PROGRAM main
  VAR
    objectDetected AT %IX0.0 : BOOL;
    heightReading AT %IW0 : INT;
    conveyorRun AT %QX0.0 : BOOL;
    diverterGate AT %QX0.1 : BOOL;
    alarmActive AT %QX0.2 : BOOL;
    startCmd AT %QX0.3 : BOOL;
    stopCmd AT %QX0.4 : BOOL;
    resetCmd AT %QX0.5 : BOOL;
    systemRunning AT %QX0.6 : BOOL;
    isTallObject : BOOL;
    TON0 : TON;
    TON1 : TON;
    h : REAL;
  END_VAR

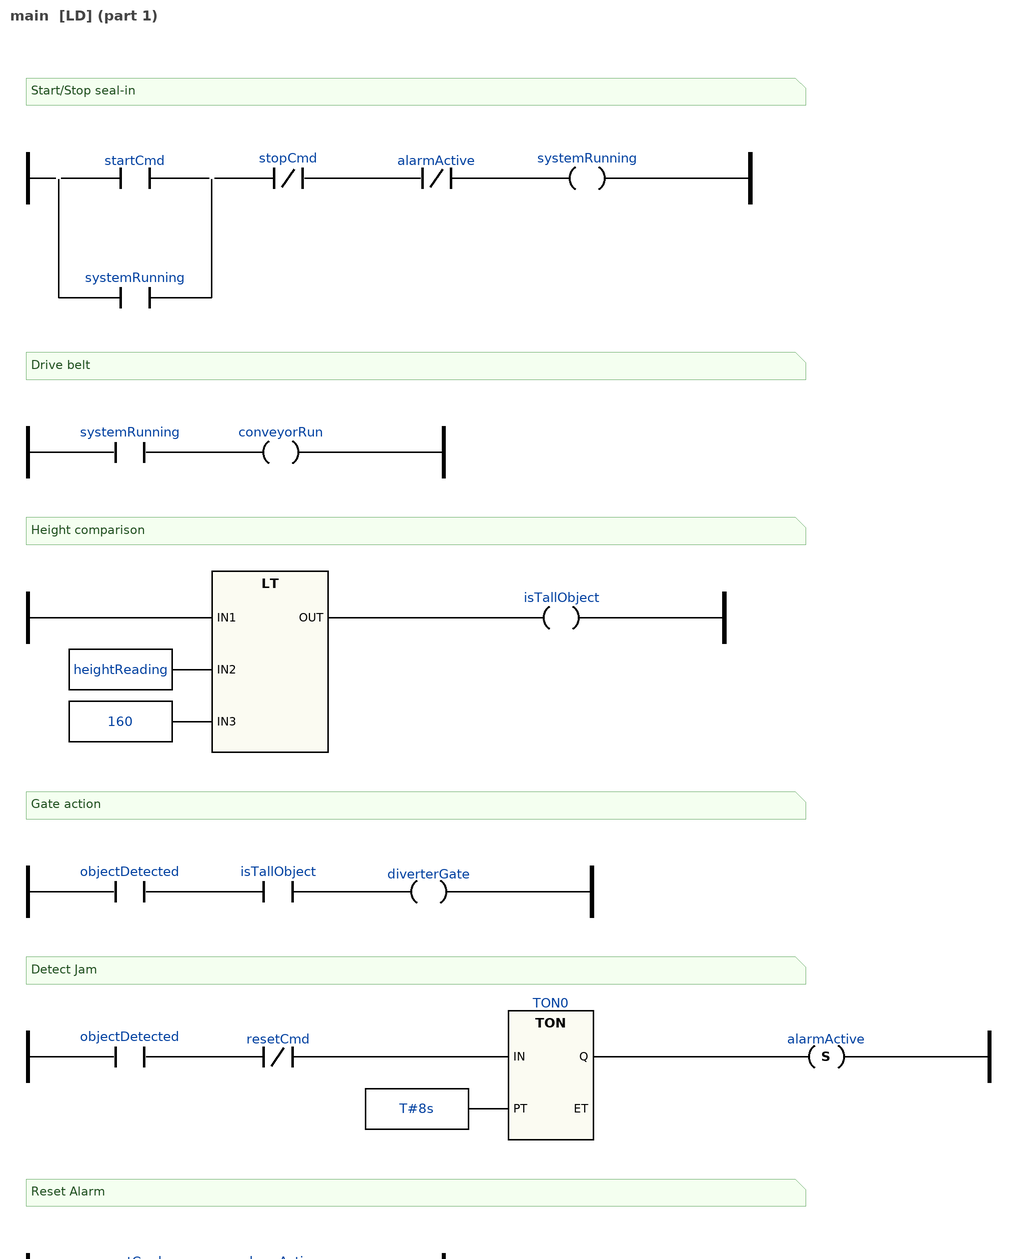
(* LD diagram, written out as Structured Text *)
(* Start/Stop seal-in *)
systemRunning := (startCmd OR systemRunning) AND NOT stopCmd AND NOT alarmActive;
(* Drive belt *)
conveyorRun := systemRunning;
(* Height comparison *)
isTallObject := LT(TRUE, heightReading, 160);
(* Gate action *)
diverterGate := objectDetected AND isTallObject;
(* Detect Jam *)
TON0(IN := objectDetected AND NOT resetCmd, PT := T#8s);
IF TON0.Q THEN alarmActive := TRUE; END_IF;
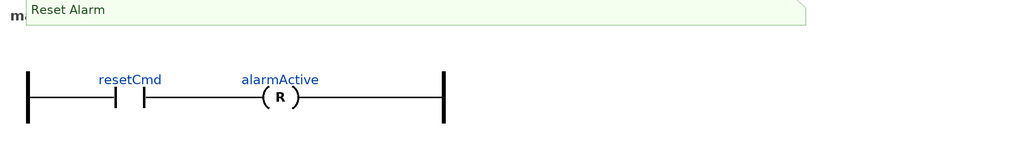
(* Reset Alarm *)
IF resetCmd THEN alarmActive := FALSE; END_IF;
END_PROGRAM
